SYSTEM Simple Test System
  (* Version 1.0, 2008-12-19, Goran Cengic, Chalmers *)
  DEVICE Test Device : DeviceType_not_used
    RESOURCE Test Resource : ResourceType_not_used
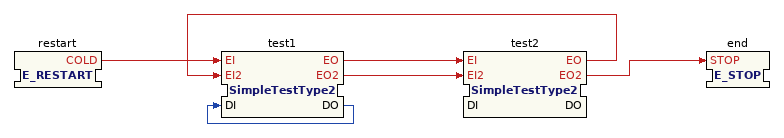
      FBS
        restart : E_RESTART;
        test1 : SimpleTestType2;
        test2 : SimpleTestType2;
        end : E_STOP;
      END_FBS
      EVENT_CONNECTIONS
        restart.COLD TO test1.EI;
        test1.EO TO test2.EI;
        test1.EO2 TO test2.EI2;
        test2.EO TO test1.EI2;
        test2.EO2 TO end.STOP;
      END_CONNECTIONS
      DATA_CONNECTIONS
        test1.DO TO test1.DI;
      END_CONNECTIONS
    END_RESOURCE
  END_DEVICE
END_SYSTEM
